// TIA Portal V17 export
// export: Created 2023-04-04T13:27:29.9876115Z, ExportSetting WithDefaults, DisplayName Totally Integrated Automation Portal, DisplayVersion V17, DisplayName TIA Portal Openness, DisplayVersion V17, DisplayName TIA Portal Version Control Interface, DisplayVersion V17, DisplayName STEP 7 Professional, DisplayVersion V17, DisplayName STEP 7 Safety, DisplayVersion V17, DisplayName WinCC Advanced, DisplayVersion V17
VAR_GLOBAL   // PLC tag table "MPO - Multi Processing Station with Oven"
   IX_MPO_RefSwitchTurnTable_PosVac_I1 AT %I1.7 : Bool;   // MPO - I1 = Reference switch turn-table (position vacuum)   {ExternalAccessible false, ExternalVisible false, ExternalWritable false}
   IX_MPO_RefSwitchTurnTable_PosBelt_I2 AT %I2.0 : Bool;   // MPO - I2 = Reference switch turn-table (position belt)   {ExternalAccessible false, ExternalVisible false, ExternalWritable false}
   IX_MPO_LightBarrierEndOfConBelt_I3 AT %I2.1 : Bool;   // MPO - I3 = Light barrier end of conveyor belt   {ExternalAccessible false, ExternalVisible false, ExternalWritable false}
   IX_MPO_RefSwitchTurnTable_PosSaw_I4 AT %I2.2 : Bool;   // MPO - I4 = Reference switch turn-table (position saw)   {ExternalAccessible false, ExternalVisible false, ExternalWritable false}
   IX_MPO_RefSwitchVac_PosTurnTable_I5 AT %I2.3 : Bool;   // MPO - I5 = Reference switch vacuum (position turn-table)   {ExternalAccessible false, ExternalVisible false, ExternalWritable false}
   IX_MPO_RefSwitchOvenFeederInside_I6 AT %I2.4 : Bool;   // MPO - I6 = Reference switch oven feeder inside   {ExternalAccessible false, ExternalVisible false, ExternalWritable false}
   IX_MPO_RefSwitchOvenFeederOutside_I7 AT %I2.5 : Bool;   // MPO - I7 = Reference switch oven feeder outside   {ExternalAccessible false, ExternalVisible false, ExternalWritable false}
   IX_MPO_RefSwitchVac_PosOven_I8 AT %I2.6 : Bool;   // MPO - I8 = Reference switch vacuum (position oven)   {ExternalAccessible false, ExternalVisible false, ExternalWritable false}
   IX_MPO_LightBarrierOven_I9 AT %I2.7 : Bool;   // MPO - I9 = Light barrier oven   {ExternalAccessible false, ExternalVisible false, ExternalWritable false}
   QX_MPO_M1_TurnTableClockwise_Q1 AT %Q3.0 : Bool;   // MPO - Q1 = Motor M1 turn-table clockwise   {ExternalAccessible false, ExternalVisible false, ExternalWritable false}
   QX_MPO_M1_TurnTableCounterclockwise_Q2 AT %Q3.1 : Bool;   // MPO - Q2 = Motor M1 turn-table counterclockwise   {ExternalAccessible false, ExternalVisible false, ExternalWritable false}
   QX_MPO_M2_ConveyorBeltForward_Q3 AT %Q3.2 : Bool;   // MPO - Q3 = Motor M2 conveyor belt forward   {ExternalAccessible false, ExternalVisible false, ExternalWritable false}
   QX_MPO_M3_Saw_Q4 AT %Q3.3 : Bool;   // MPO - Q4 = Motor M3 saw   {ExternalAccessible false, ExternalVisible false, ExternalWritable false}
   QX_MPO_M4_OvenFeederRetract_Q5 AT %Q3.4 : Bool;   // MPO - Q5 = Motor M4 oven feeder retract   {ExternalAccessible false, ExternalVisible false, ExternalWritable false}
   QX_MPO_M4_OvenFeederExtend_Q6 AT %Q3.5 : Bool;   // MPO - Q6 = Motor M4 oven feeder extend   {ExternalAccessible false, ExternalVisible false, ExternalWritable false}
   QX_MPO_M5_VacuumTowardsOven_Q7 AT %Q3.6 : Bool;   // MPO - Q7 = Motor M5 vacuum towards oven   {ExternalAccessible false, ExternalVisible false, ExternalWritable false}
   QX_MPO_M5_VacuumTowardsTurnTable_Q8 AT %Q3.7 : Bool;   // MPO - Q8 = Motor M5 vacuum towards turn-table   {ExternalAccessible false, ExternalVisible false, ExternalWritable false}
   QX_MPO_LightOven_Q9 AT %Q4.0 : Bool;   // MPO - Q9 = Light oven   {ExternalAccessible false, ExternalVisible false, ExternalWritable false}
   QX_MPO_Compressor_Q10 AT %Q4.1 : Bool;   // MPO - Q10 = Compressor   {ExternalAccessible false, ExternalVisible false, ExternalWritable false}
   QX_MPO_ValveVacuum_Q11 AT %Q4.2 : Bool;   // MPO - Q11 = Valve vacuum   {ExternalAccessible false, ExternalVisible false, ExternalWritable false}
   QX_MPO_ValveLowering_Q12 AT %Q4.3 : Bool;   // MPO - Q12 = Valve lowering   {ExternalAccessible false, ExternalVisible false, ExternalWritable false}
   QX_MPO_ValveOvenDoor_Q13 AT %Q4.4 : Bool;   // MPO - Q13 = Valve oven door   {ExternalAccessible false, ExternalVisible false, ExternalWritable false}
   QX_MPO_ValveFeeder_Q14 AT %Q4.5 : Bool;   // MPO - Q14 = Valve feeder   {ExternalAccessible false, ExternalVisible false, ExternalWritable false}
   QW_MPO_PWM_TurnTable_M1 AT %QW23 : Int;   // MPO = PWM Motor M1 turn-table   {ExternalAccessible false, ExternalVisible false, ExternalWritable false}
   QW_MPO_PWM_Vacuum_M5 AT %QW25 : Int;   // MPO = PWM Motor M5 vacuum   {ExternalAccessible false, ExternalVisible false, ExternalWritable false}
END_VAR
